KUKA KRL program: FOLGE7.SRC, FOLGE7.DAT

--- FOLGE7.SRC ---
&COMMENT vymena cepicek
&ACCESS RV
&PARAM TPVW_VERSION=3.3.5
DEF FOLGE7 ( )
; FOLD ;%{H} %MKUKATPVW
SPS_N=-1
VW (#VW_AUE_INIT,TRUE)
PENTER:
INTERRUPT DECL 10 WHEN $CYCFLAG[30]==FALSE DO VW(#FB_STOP,TRUE)
INTERRUPT ON 10
INT10=TRUE
; ENDFOLD
;FOLD PTP VB=100% VE=0% ACC=100% Wzg=1 SPSTrig=0[1/100s] FP;%{P}%MKUKATPVW,%CMOVE,%VPTP,%P 1:1, 2: VB=, 3:100, 4:%, 5: VE=, 6:0, 7:%, 8: ACC=, 9:100, 10:%, 11: Wzg=, 12:1, 13: SPSTrig=, 14:0, 15:[1/100s], 16: FP, 17:0, 18:-1, 19:1
; FOLD FB ONL = EIN;%{SE}%MKUKATPVW %CVW_SPS %VFB %P 2:FB ONL = EIN,3:                  FB
;ENDFOLD
;FOLD 1:  SPSMAKRO99 = !F100;%{SE}%MKUKATPVW %CVW_SPS %VMAKRO %P 2:SPSMAKRO99 = !F100,3:             MAKRO
;ENDFOLD
;FOLD 2:  SPSMAKRO96 = EIN;%{SE}%MKUKATPVW %CVW_SPS %VMAKRO %P 2:SPSMAKRO96 = EIN,3:               MAKRO
;ENDFOLD
;FOLD 3:  SPSMAKRO81 = EIN;%{SE}%MKUKATPVW %CVW_SPS %VMAKRO %P 2:SPSMAKRO81 = EIN,3:            MAKRO
;ENDFOLD
;FOLD 4:  SPSMAKRO82 = EIN;%{SE}%MKUKATPVW %CVW_SPS %VMAKRO %P 2:SPSMAKRO82 = EIN,3:           MAKRO
;ENDFOLD
;FOLD 5:  SPSMAKRO95 = EIN;%{SE}%MKUKATPVW %CVW_SPS %VMAKRO %P 2:SPSMAKRO95 = EIN,3:                 MAKRO
;ENDFOLD
;FOLD 6:  bin1 ( EIN ) = 9931;%{SE}%MKUKATPVW %CVW_SPS %VARIASG %P 2:bin1 ( EIN ) = 9931,3:          ARIASG
;ENDFOLD
;FOLD 7:  SPSMAKRO3 = EIN;%{SE}%MKUKATPVW %CVW_SPS %VMAKRO %P 2:SPSMAKRO3 = EIN,3:         MAKRO
;ENDFOLD
;FOLD {H}
SPS_FERTIG = FALSE
INTERRUPT DECL 10 WHEN $CYCFLAG[30]==FALSE DO VW(#FB_STOP,TRUE)
INTERRUPT ON 10
INT10=TRUE
VW(#VW_INIT,TRUE)
VW_USR_R (#USR_INIT)
TRIGGER  WHEN DISTANCE=1 DELAY=-0.1 DO P0_MERKER=TRUE
VW_MPARA_ACT = P0_D
VW(#MPARA,TRUE)
SPS_FERTIG=FALSE
TRIGGER WHEN DISTANCE=1 DELAY=0 DO SPS_TRIG(1) PRIO=-1
TRIGGER WHEN DISTANCE=0 DELAY=0 DO $CYCFLAG[30]=(TRUE) AND $CYCFLAG[31] OR ($TIMER[15]<0)
TRIGGER WHEN DISTANCE=0 DELAY=0 DO $CYC_DEF30[]=" EIN "
PTP P0
WAIT FOR SPS_FERTIG
;ENDFOLD
;ENDFOLD
; FOLD Warte auf Folgenstart ;%{SE}%MKUKATPVW,%C,%V
VW (#VW_AUE_WAIT,TRUE )
IF N_VW==TRUE THEN
GOTO PEXIT
ENDIF
;ENDFOLD
;FOLD PTP VB=100% VE=0% ACC=100% Wzg=1 SPSTrig=0[1/100s] FP;%{P}%MKUKATPVW,%CMOVE,%VPTP,%P 1:1, 2: VB=, 3:100, 4:%, 5: VE=, 6:0, 7:%, 8: ACC=, 9:100, 10:%, 11: Wzg=, 12:1, 13: SPSTrig=, 14:0, 15:[1/100s], 16: FP, 17:1, 18:-1, 19:2
; FOLD FB ONL = EIN;%{SE}%MKUKATPVW %CVW_SPS %VFB %P 2:FB ONL = EIN,3:           FB
;ENDFOLD
;FOLD 1:  F100 = AUS;%{SE}%MKUKATPVW %CVW_SPS %VBOASG %P 2:F100 = AUS,3:          BOASG
;ENDFOLD
;FOLD 2:  F199 = EIN;%{SE}%MKUKATPVW %CVW_SPS %VBOASG %P 2:F199 = EIN,3:         BOASG
;ENDFOLD
;FOLD 3:  SPSMAKRO21 = EIN;%{SE}%MKUKATPVW %CVW_SPS %VMAKRO %P 2:SPSMAKRO21 = EIN,3:        MAKRO
;ENDFOLD
;FOLD 4:  t1 ( EIN ) = 0[1/10Sek];%{SE}%MKUKATPVW %CVW_SPS %VTASG %P 2:t1 ( EIN ) = 0[1/10Sek],3:       TASG
;ENDFOLD
;FOLD {H}
VW_MPARA_ACT = P1_D
VW(#MPARA,TRUE)
SPS_FERTIG=FALSE
TRIGGER WHEN DISTANCE=1 DELAY=0 DO SPS_TRIG(2) PRIO=-1
TRIGGER WHEN DISTANCE=0 DELAY=0 DO $CYCFLAG[30]=(TRUE) AND $CYCFLAG[31] OR ($TIMER[15]<0)
TRIGGER WHEN DISTANCE=0 DELAY=0 DO $CYC_DEF30[]=" EIN "
PTP P1
WAIT FOR SPS_FERTIG
;ENDFOLD
;ENDFOLD
;FOLD PTP VB=100% VE=0% ACC=100% Wzg=1 SPSTrig=0[1/100s] FU;%{P}%MKUKATPVW,%CMOVE,%VPTP,%P 1:1, 2: VB=, 3:100, 4:%, 5: VE=, 6:0, 7:%, 8: ACC=, 9:100, 10:%, 11: Wzg=, 12:1, 13: SPSTrig=, 14:0, 15:[1/100s], 16: FU, 17:3, 18:-1, 19:-1
; FOLD FB ONL = M1;%{SE}%MKUKATPVW %CVW_SPS %VFB %P 2:FB ONL = M1,3:          FB
;ENDFOLD
; FOLD UP8 = F409;%{SE}%MKUKATPVW %CVW_SPS %VUP %P 2:UP8 = F409,3:       UP
;ENDFOLD
; FOLD UP1 = E67 + F401;%{SE}%MKUKATPVW %CVW_SPS %VUP %P 2:UP1 = E67 + F401,3:        UP
;ENDFOLD
;FOLD {H}
VW_MPARA_ACT = P3_D
VW(#MPARA,TRUE)
TRIGGER WHEN DISTANCE=0 DELAY=0 DO $CYCFLAG[30]=($CYCFLAG[1]) AND $CYCFLAG[31] OR ($TIMER[15]<0)
TRIGGER WHEN DISTANCE=0 DELAY=0 DO $CYC_DEF30[]="M1"
PTP P3
WAIT FOR TRUE
SELECT(#UP,8,$FLAG[409])
SELECT(#UP,1,$IN[67] OR $FLAG[401])
;ENDFOLD
;ENDFOLD
;FOLD PTP VB=100% VE=0% ACC=100% Wzg=1 SPSTrig=0[1/100s] FP;%{P}%MKUKATPVW,%CMOVE,%VPTP,%P 1:1, 2: VB=, 3:100, 4:%, 5: VE=, 6:0, 7:%, 8: ACC=, 9:100, 10:%, 11: Wzg=, 12:1, 13: SPSTrig=, 14:0, 15:[1/100s], 16: FP, 17:2, 18:-1, 19:3
; FOLD FB ONL = EIN;%{SE}%MKUKATPVW %CVW_SPS %VFB %P 2:FB ONL = EIN,3:             FB
;ENDFOLD
;FOLD 1:  F100 = EIN;%{SE}%MKUKATPVW %CVW_SPS %VBOASG %P 2:F100 = EIN,3:            BOASG
;ENDFOLD
;FOLD 2:  F199 = AUS;%{SE}%MKUKATPVW %CVW_SPS %VBOASG %P 2:F199 = AUS,3:         BOASG
;ENDFOLD
;FOLD 3:  t1 ( EIN ) = STOP;%{SE}%MKUKATPVW %CVW_SPS %VTSTOP %P 2:t1 ( EIN ) = STOP,3:        TSTOP
;ENDFOLD
;FOLD 4:  t2 ( EIN ) = t1[1/10Sek];%{SE}%MKUKATPVW %CVW_SPS %VTASG %P 2:t2 ( EIN ) = t1[1/10Sek],3:        TASG
;ENDFOLD
;FOLD 5:  t2 ( EIN ) = STOP;%{SE}%MKUKATPVW %CVW_SPS %VTSTOP %P 2:t2 ( EIN ) = STOP,3:       TSTOP
;ENDFOLD
;FOLD 6:  SPSMAKRO81 = EIN;%{SE}%MKUKATPVW %CVW_SPS %VMAKRO %P 2:SPSMAKRO81 = EIN,3:           MAKRO
;ENDFOLD
;FOLD 7:  SPSMAKRO82 = EIN;%{SE}%MKUKATPVW %CVW_SPS %VMAKRO %P 2:SPSMAKRO82 = EIN,3:          MAKRO
;ENDFOLD
;FOLD {H}
VW_MPARA_ACT = P2_D
VW(#MPARA,TRUE)
SPS_FERTIG=FALSE
TRIGGER WHEN DISTANCE=1 DELAY=0 DO SPS_TRIG(3) PRIO=-1
TRIGGER WHEN DISTANCE=0 DELAY=0 DO $CYCFLAG[30]=(TRUE) AND $CYCFLAG[31] OR ($TIMER[15]<0)
TRIGGER WHEN DISTANCE=0 DELAY=0 DO $CYC_DEF30[]=" EIN "
PTP P2
WAIT FOR SPS_FERTIG
;ENDFOLD
;ENDFOLD
; FOLD ;%{H}
VW (#VW_AUE_END,TRUE)
GOTO PENTER
PEXIT:
END
DEF  SPS_TRIG (NO:IN )
INT NO
BOOL UES
IF NO>10000 THEN
NO=NO-10000
UES=TRUE
ELSE
UES=FALSE
ENDIF
IF $PRO_MODE==#MSTEP THEN
IF $PRO_MOVE THEN
WAIT FOR NOT $PRO_MOVE
HALT
ENDIF
ENDIF
SWITCH  NO
CASE 1
;FOLD SPS_TRIG1 {H}
SELECT(#MAKRO,99,NOT $FLAG[100])
SELECT(#MAKRO,96,TRUE)
SELECT(#MAKRO,81,TRUE)
SELECT(#MAKRO,82,TRUE)
SELECT(#MAKRO,95,TRUE)
VW(#BINOUT,TRUE,1,9931)
SELECT(#MAKRO,3,TRUE)
;ENDFOLD
CASE 2
;FOLD SPS_TRIG2 {H}
$FLAG[100]=FALSE
$FLAG[199]=TRUE
SELECT(#MAKRO,21,TRUE)
VW(#SET_TIME,TRUE,1,0,0)
;ENDFOLD
CASE 3
;FOLD SPS_TRIG3 {H}
$FLAG[100]=TRUE
$FLAG[199]=FALSE
VW(#SET_TIME,TRUE,1,1,0)
VW(#SET_TIME,TRUE,2,0,$TIMER[1]*0.01)
VW(#SET_TIME,TRUE,2,1,0)
SELECT(#MAKRO,81,TRUE)
SELECT(#MAKRO,82,TRUE)
;ENDFOLD
CASE 4
;FOLD SPS_TRIG4 {H}
;ENDFOLD
CASE 5
;FOLD SPS_TRIG5 {H}
;ENDFOLD
CASE 6
;FOLD SPS_TRIG6 {H}
;ENDFOLD
CASE 7
;FOLD SPS_TRIG7 {H}
;ENDFOLD
CASE 8
;FOLD SPS_TRIG8 {H}
;ENDFOLD
CASE 9
;FOLD SPS_TRIG9 {H}
;ENDFOLD
CASE 10
;FOLD SPS_TRIG10 {H}
;ENDFOLD
CASE 11
;FOLD SPS_TRIG11 {H}
;ENDFOLD
CASE 12
;FOLD SPS_TRIG12 {H}
;ENDFOLD
CASE 13
;FOLD SPS_TRIG13 {H}
;ENDFOLD
CASE 14
;FOLD SPS_TRIG14 {H}
;ENDFOLD
CASE 15
;FOLD SPS_TRIG15 {H}
;ENDFOLD
CASE 16
;FOLD SPS_TRIG16 {H}
;ENDFOLD
CASE 17
;FOLD SPS_TRIG17 {H}
;ENDFOLD
CASE 18
;FOLD SPS_TRIG18 {H}
;ENDFOLD
CASE 19
;FOLD SPS_TRIG19 {H}
;ENDFOLD
CASE 20
;FOLD SPS_TRIG20 {H}
;ENDFOLD
CASE 21
;FOLD SPS_TRIG21 {H}
;ENDFOLD
CASE 22
;FOLD SPS_TRIG22 {H}
;ENDFOLD
CASE 23
;FOLD SPS_TRIG23 {H}
;ENDFOLD
CASE 24
;FOLD SPS_TRIG24 {H}
;ENDFOLD
CASE 25
;FOLD SPS_TRIG25 {H}
;ENDFOLD
CASE 26
;FOLD SPS_TRIG26 {H}
;ENDFOLD
CASE 27
;FOLD SPS_TRIG27 {H}
;ENDFOLD
CASE 28
;FOLD SPS_TRIG28 {H}
;ENDFOLD
CASE 29
;FOLD SPS_TRIG29 {H}
;ENDFOLD
CASE 30
;FOLD SPS_TRIG30 {H}
;ENDFOLD
CASE 31
;FOLD SPS_TRIG31 {H}
;ENDFOLD
CASE 32
;FOLD SPS_TRIG32 {H}
;ENDFOLD
CASE 33
;FOLD SPS_TRIG33 {H}
;ENDFOLD
CASE 34
;FOLD SPS_TRIG34 {H}
;ENDFOLD
CASE 35
;FOLD SPS_TRIG35 {H}
;ENDFOLD
CASE 36
;FOLD SPS_TRIG36 {H}
;ENDFOLD
CASE 37
;FOLD SPS_TRIG37 {H}
;ENDFOLD
CASE 38
;FOLD SPS_TRIG38 {H}
;ENDFOLD
CASE 39
;FOLD SPS_TRIG39 {H}
;ENDFOLD
CASE 40
;FOLD SPS_TRIG40 {H}
;ENDFOLD
CASE 41
;FOLD SPS_TRIG41 {H}
;ENDFOLD
CASE 42
;FOLD SPS_TRIG42 {H}
;ENDFOLD
CASE 43
;FOLD SPS_TRIG43 {H}
;ENDFOLD
CASE 44
;FOLD SPS_TRIG44 {H}
;ENDFOLD
CASE 45
;FOLD SPS_TRIG45 {H}
;ENDFOLD
CASE 46
;FOLD SPS_TRIG46 {H}
;ENDFOLD
CASE 47
;FOLD SPS_TRIG47 {H}
;ENDFOLD
CASE 48
;FOLD SPS_TRIG48 {H}
;ENDFOLD
CASE 49
;FOLD SPS_TRIG49 {H}
;ENDFOLD
CASE 50
;FOLD SPS_TRIG50 {H}
;ENDFOLD
CASE 51
;FOLD SPS_TRIG51 {H}
;ENDFOLD
CASE 52
;FOLD SPS_TRIG52 {H}
;ENDFOLD
CASE 53
;FOLD SPS_TRIG53 {H}
;ENDFOLD
CASE 54
;FOLD SPS_TRIG54 {H}
;ENDFOLD
CASE 55
;FOLD SPS_TRIG55 {H}
;ENDFOLD
CASE 56
;FOLD SPS_TRIG56 {H}
;ENDFOLD
CASE 57
;FOLD SPS_TRIG57 {H}
;ENDFOLD
CASE 58
;FOLD SPS_TRIG58 {H}
;ENDFOLD
CASE 59
;FOLD SPS_TRIG59 {H}
;ENDFOLD
CASE 60
;FOLD SPS_TRIG60 {H}
;ENDFOLD
CASE 61
;FOLD SPS_TRIG61 {H}
;ENDFOLD
CASE 62
;FOLD SPS_TRIG62 {H}
;ENDFOLD
CASE 63
;FOLD SPS_TRIG63 {H}
;ENDFOLD
CASE 64
;FOLD SPS_TRIG64 {H}
;ENDFOLD
CASE 65
;FOLD SPS_TRIG65 {H}
;ENDFOLD
CASE 66
;FOLD SPS_TRIG66 {H}
;ENDFOLD
CASE 67
;FOLD SPS_TRIG67 {H}
;ENDFOLD
CASE 68
;FOLD SPS_TRIG68 {H}
;ENDFOLD
CASE 69
;FOLD SPS_TRIG69 {H}
;ENDFOLD
CASE 70
;FOLD SPS_TRIG70 {H}
;ENDFOLD
CASE 71
;FOLD SPS_TRIG71 {H}
;ENDFOLD
CASE 72
;FOLD SPS_TRIG72 {H}
;ENDFOLD
CASE 73
;FOLD SPS_TRIG73 {H}
;ENDFOLD
CASE 74
;FOLD SPS_TRIG74 {H}
;ENDFOLD
CASE 75
;FOLD SPS_TRIG75 {H}
;ENDFOLD
CASE 76
;FOLD SPS_TRIG76 {H}
;ENDFOLD
CASE 77
;FOLD SPS_TRIG77 {H}
;ENDFOLD
CASE 78
;FOLD SPS_TRIG78 {H}
;ENDFOLD
CASE 79
;FOLD SPS_TRIG79 {H}
;ENDFOLD
CASE 80
;FOLD SPS_TRIG80 {H}
;ENDFOLD
CASE 81
;FOLD SPS_TRIG81 {H}
;ENDFOLD
CASE 82
;FOLD SPS_TRIG82 {H}
;ENDFOLD
CASE 83
;FOLD SPS_TRIG83 {H}
;ENDFOLD
CASE 84
;FOLD SPS_TRIG84 {H}
;ENDFOLD
CASE 85
;FOLD SPS_TRIG85 {H}
;ENDFOLD
CASE 86
;FOLD SPS_TRIG86 {H}
;ENDFOLD
CASE 87
;FOLD SPS_TRIG87 {H}
;ENDFOLD
CASE 88
;FOLD SPS_TRIG88 {H}
;ENDFOLD
CASE 89
;FOLD SPS_TRIG89 {H}
;ENDFOLD
CASE 90
;FOLD SPS_TRIG90 {H}
;ENDFOLD
CASE 91
;FOLD SPS_TRIG91 {H}
;ENDFOLD
CASE 92
;FOLD SPS_TRIG92 {H}
;ENDFOLD
CASE 93
;FOLD SPS_TRIG93 {H}
;ENDFOLD
CASE 94
;FOLD SPS_TRIG94 {H}
;ENDFOLD
CASE 95
;FOLD SPS_TRIG95 {H}
;ENDFOLD
CASE 96
;FOLD SPS_TRIG96 {H}
;ENDFOLD
CASE 97
;FOLD SPS_TRIG97 {H}
;ENDFOLD
CASE 98
;FOLD SPS_TRIG98 {H}
;ENDFOLD
CASE 99
;FOLD SPS_TRIG99 {H}
;ENDFOLD
CASE 100
;FOLD SPS_TRIG100 {H}
;ENDFOLD
CASE 101
;FOLD SPS_TRIG101 {H}
;ENDFOLD
CASE 102
;FOLD SPS_TRIG102 {H}
;ENDFOLD
CASE 103
;FOLD SPS_TRIG103 {H}
;ENDFOLD
CASE 104
;FOLD SPS_TRIG104 {H}
;ENDFOLD
CASE 105
;FOLD SPS_TRIG105 {H}
;ENDFOLD
CASE 106
;FOLD SPS_TRIG106 {H}
;ENDFOLD
CASE 107
;FOLD SPS_TRIG107 {H}
;ENDFOLD
CASE 108
;FOLD SPS_TRIG108 {H}
;ENDFOLD
CASE 109
;FOLD SPS_TRIG109 {H}
;ENDFOLD
CASE 110
;FOLD SPS_TRIG110 {H}
;ENDFOLD
CASE 111
;FOLD SPS_TRIG111 {H}
;ENDFOLD
CASE 112
;FOLD SPS_TRIG112 {H}
;ENDFOLD
CASE 113
;FOLD SPS_TRIG113 {H}
;ENDFOLD
CASE 114
;FOLD SPS_TRIG114 {H}
;ENDFOLD
CASE 115
;FOLD SPS_TRIG115 {H}
;ENDFOLD
CASE 116
;FOLD SPS_TRIG116 {H}
;ENDFOLD
CASE 117
;FOLD SPS_TRIG117 {H}
;ENDFOLD
CASE 118
;FOLD SPS_TRIG118 {H}
;ENDFOLD
CASE 119
;FOLD SPS_TRIG119 {H}
;ENDFOLD
CASE 120
;FOLD SPS_TRIG120 {H}
;ENDFOLD
CASE 121
;FOLD SPS_TRIG121 {H}
;ENDFOLD
CASE 122
;FOLD SPS_TRIG122 {H}
;ENDFOLD
CASE 123
;FOLD SPS_TRIG123 {H}
;ENDFOLD
CASE 124
;FOLD SPS_TRIG124 {H}
;ENDFOLD
CASE 125
;FOLD SPS_TRIG125 {H}
;ENDFOLD
CASE 126
;FOLD SPS_TRIG126 {H}
;ENDFOLD
CASE 127
;FOLD SPS_TRIG127 {H}
;ENDFOLD
CASE 128
;FOLD SPS_TRIG128 {H}
;ENDFOLD
CASE 129
;FOLD SPS_TRIG129 {H}
;ENDFOLD
CASE 130
;FOLD SPS_TRIG130 {H}
;ENDFOLD
CASE 131
;FOLD SPS_TRIG131 {H}
;ENDFOLD
CASE 132
;FOLD SPS_TRIG132 {H}
;ENDFOLD
CASE 133
;FOLD SPS_TRIG133 {H}
;ENDFOLD
CASE 134
;FOLD SPS_TRIG134 {H}
;ENDFOLD
CASE 135
;FOLD SPS_TRIG135 {H}
;ENDFOLD
CASE 136
;FOLD SPS_TRIG136 {H}
;ENDFOLD
CASE 137
;FOLD SPS_TRIG137 {H}
;ENDFOLD
CASE 138
;FOLD SPS_TRIG138 {H}
;ENDFOLD
CASE 139
;FOLD SPS_TRIG139 {H}
;ENDFOLD
CASE 140
;FOLD SPS_TRIG140 {H}
;ENDFOLD
CASE 141
;FOLD SPS_TRIG141 {H}
;ENDFOLD
CASE 142
;FOLD SPS_TRIG142 {H}
;ENDFOLD
CASE 143
;FOLD SPS_TRIG143 {H}
;ENDFOLD
CASE 144
;FOLD SPS_TRIG144 {H}
;ENDFOLD
CASE 145
;FOLD SPS_TRIG145 {H}
;ENDFOLD
CASE 146
;FOLD SPS_TRIG146 {H}
;ENDFOLD
CASE 147
;FOLD SPS_TRIG147 {H}
;ENDFOLD
CASE 148
;FOLD SPS_TRIG148 {H}
;ENDFOLD
CASE 149
;FOLD SPS_TRIG149 {H}
;ENDFOLD
CASE 150
;FOLD SPS_TRIG150 {H}
;ENDFOLD
CASE 151
;FOLD SPS_TRIG151 {H}
;ENDFOLD
CASE 152
;FOLD SPS_TRIG152 {H}
;ENDFOLD
CASE 153
;FOLD SPS_TRIG153 {H}
;ENDFOLD
CASE 154
;FOLD SPS_TRIG154 {H}
;ENDFOLD
CASE 155
;FOLD SPS_TRIG155 {H}
;ENDFOLD
CASE 156
;FOLD SPS_TRIG156 {H}
;ENDFOLD
CASE 157
;FOLD SPS_TRIG157 {H}
;ENDFOLD
CASE 158
;FOLD SPS_TRIG158 {H}
;ENDFOLD
CASE 159
;FOLD SPS_TRIG159 {H}
;ENDFOLD
CASE 160
;FOLD SPS_TRIG160 {H}
;ENDFOLD
CASE 161
;FOLD SPS_TRIG161 {H}
;ENDFOLD
CASE 162
;FOLD SPS_TRIG162 {H}
;ENDFOLD
CASE 163
;FOLD SPS_TRIG163 {H}
;ENDFOLD
CASE 164
;FOLD SPS_TRIG164 {H}
;ENDFOLD
CASE 165
;FOLD SPS_TRIG165 {H}
;ENDFOLD
CASE 166
;FOLD SPS_TRIG166 {H}
;ENDFOLD
CASE 167
;FOLD SPS_TRIG167 {H}
;ENDFOLD
CASE 168
;FOLD SPS_TRIG168 {H}
;ENDFOLD
CASE 169
;FOLD SPS_TRIG169 {H}
;ENDFOLD
CASE 170
;FOLD SPS_TRIG170 {H}
;ENDFOLD
CASE 171
;FOLD SPS_TRIG171 {H}
;ENDFOLD
CASE 172
;FOLD SPS_TRIG172 {H}
;ENDFOLD
CASE 173
;FOLD SPS_TRIG173 {H}
;ENDFOLD
CASE 174
;FOLD SPS_TRIG174 {H}
;ENDFOLD
CASE 175
;FOLD SPS_TRIG175 {H}
;ENDFOLD
CASE 176
;FOLD SPS_TRIG176 {H}
;ENDFOLD
CASE 177
;FOLD SPS_TRIG177 {H}
;ENDFOLD
CASE 178
;FOLD SPS_TRIG178 {H}
;ENDFOLD
CASE 179
;FOLD SPS_TRIG179 {H}
;ENDFOLD
CASE 180
;FOLD SPS_TRIG180 {H}
;ENDFOLD
CASE 181
;FOLD SPS_TRIG181 {H}
;ENDFOLD
CASE 182
;FOLD SPS_TRIG182 {H}
;ENDFOLD
CASE 183
;FOLD SPS_TRIG183 {H}
;ENDFOLD
CASE 184
;FOLD SPS_TRIG184 {H}
;ENDFOLD
CASE 185
;FOLD SPS_TRIG185 {H}
;ENDFOLD
CASE 186
;FOLD SPS_TRIG186 {H}
;ENDFOLD
CASE 187
;FOLD SPS_TRIG187 {H}
;ENDFOLD
CASE 188
;FOLD SPS_TRIG188 {H}
;ENDFOLD
CASE 189
;FOLD SPS_TRIG189 {H}
;ENDFOLD
CASE 190
;FOLD SPS_TRIG190 {H}
;ENDFOLD
CASE 191
;FOLD SPS_TRIG191 {H}
;ENDFOLD
CASE 192
;FOLD SPS_TRIG192 {H}
;ENDFOLD
CASE 193
;FOLD SPS_TRIG193 {H}
;ENDFOLD
CASE 194
;FOLD SPS_TRIG194 {H}
;ENDFOLD
CASE 195
;FOLD SPS_TRIG195 {H}
;ENDFOLD
CASE 196
;FOLD SPS_TRIG196 {H}
;ENDFOLD
CASE 197
;FOLD SPS_TRIG197 {H}
;ENDFOLD
CASE 198
;FOLD SPS_TRIG198 {H}
;ENDFOLD
CASE 199
;FOLD SPS_TRIG199 {H}
;ENDFOLD
CASE 200
;FOLD SPS_TRIG200 {H}
;ENDFOLD
CASE 201
;FOLD SPS_TRIG201 {H}
;ENDFOLD
CASE 202
;FOLD SPS_TRIG202 {H}
;ENDFOLD
CASE 203
;FOLD SPS_TRIG203 {H}
;ENDFOLD
CASE 204
;FOLD SPS_TRIG204 {H}
;ENDFOLD
CASE 205
;FOLD SPS_TRIG205 {H}
;ENDFOLD
CASE 206
;FOLD SPS_TRIG206 {H}
;ENDFOLD
CASE 207
;FOLD SPS_TRIG207 {H}
;ENDFOLD
CASE 208
;FOLD SPS_TRIG208 {H}
;ENDFOLD
CASE 209
;FOLD SPS_TRIG209 {H}
;ENDFOLD
CASE 210
;FOLD SPS_TRIG210 {H}
;ENDFOLD
CASE 211
;FOLD SPS_TRIG211 {H}
;ENDFOLD
CASE 212
;FOLD SPS_TRIG212 {H}
;ENDFOLD
CASE 213
;FOLD SPS_TRIG213 {H}
;ENDFOLD
CASE 214
;FOLD SPS_TRIG214 {H}
;ENDFOLD
CASE 215
;FOLD SPS_TRIG215 {H}
;ENDFOLD
CASE 216
;FOLD SPS_TRIG216 {H}
;ENDFOLD
CASE 217
;FOLD SPS_TRIG217 {H}
;ENDFOLD
CASE 218
;FOLD SPS_TRIG218 {H}
;ENDFOLD
CASE 219
;FOLD SPS_TRIG219 {H}
;ENDFOLD
CASE 220
;FOLD SPS_TRIG220 {H}
;ENDFOLD
CASE 221
;FOLD SPS_TRIG221 {H}
;ENDFOLD
CASE 222
;FOLD SPS_TRIG222 {H}
;ENDFOLD
CASE 223
;FOLD SPS_TRIG223 {H}
;ENDFOLD
CASE 224
;FOLD SPS_TRIG224 {H}
;ENDFOLD
CASE 225
;FOLD SPS_TRIG225 {H}
;ENDFOLD
CASE 226
;FOLD SPS_TRIG226 {H}
;ENDFOLD
CASE 227
;FOLD SPS_TRIG227 {H}
;ENDFOLD
CASE 228
;FOLD SPS_TRIG228 {H}
;ENDFOLD
CASE 229
;FOLD SPS_TRIG229 {H}
;ENDFOLD
CASE 230
;FOLD SPS_TRIG230 {H}
;ENDFOLD
CASE 231
;FOLD SPS_TRIG231 {H}
;ENDFOLD
CASE 232
;FOLD SPS_TRIG232 {H}
;ENDFOLD
CASE 233
;FOLD SPS_TRIG233 {H}
;ENDFOLD
CASE 234
;FOLD SPS_TRIG234 {H}
;ENDFOLD
CASE 235
;FOLD SPS_TRIG235 {H}
;ENDFOLD
CASE 236
;FOLD SPS_TRIG236 {H}
;ENDFOLD
CASE 237
;FOLD SPS_TRIG237 {H}
;ENDFOLD
CASE 238
;FOLD SPS_TRIG238 {H}
;ENDFOLD
CASE 239
;FOLD SPS_TRIG239 {H}
;ENDFOLD
CASE 240
;FOLD SPS_TRIG240 {H}
;ENDFOLD
CASE 241
;FOLD SPS_TRIG241 {H}
;ENDFOLD
CASE 242
;FOLD SPS_TRIG242 {H}
;ENDFOLD
CASE 243
;FOLD SPS_TRIG243 {H}
;ENDFOLD
CASE 244
;FOLD SPS_TRIG244 {H}
;ENDFOLD
CASE 245
;FOLD SPS_TRIG245 {H}
;ENDFOLD
CASE 246
;FOLD SPS_TRIG246 {H}
;ENDFOLD
CASE 247
;FOLD SPS_TRIG247 {H}
;ENDFOLD
CASE 248
;FOLD SPS_TRIG248 {H}
;ENDFOLD
CASE 249
;FOLD SPS_TRIG249 {H}
;ENDFOLD
CASE 250
;FOLD SPS_TRIG250 {H}
;ENDFOLD
CASE 251
;FOLD SPS_TRIG251 {H}
;ENDFOLD
CASE 252
;FOLD SPS_TRIG252 {H}
;ENDFOLD
CASE 253
;FOLD SPS_TRIG253 {H}
;ENDFOLD
CASE 254
;FOLD SPS_TRIG254 {H}
;ENDFOLD
CASE 255
;FOLD SPS_TRIG255 {H}
;ENDFOLD
CASE 256
;FOLD SPS_TRIG256 {H}
;ENDFOLD
CASE 257
;FOLD SPS_TRIG257 {H}
;ENDFOLD
CASE 258
;FOLD SPS_TRIG258 {H}
;ENDFOLD
CASE 259
;FOLD SPS_TRIG259 {H}
;ENDFOLD
CASE 260
;FOLD SPS_TRIG260 {H}
;ENDFOLD
CASE 261
;FOLD SPS_TRIG261 {H}
;ENDFOLD
CASE 262
;FOLD SPS_TRIG262 {H}
;ENDFOLD
CASE 263
;FOLD SPS_TRIG263 {H}
;ENDFOLD
CASE 264
;FOLD SPS_TRIG264 {H}
;ENDFOLD
CASE 265
;FOLD SPS_TRIG265 {H}
;ENDFOLD
CASE 266
;FOLD SPS_TRIG266 {H}
;ENDFOLD
CASE 267
;FOLD SPS_TRIG267 {H}
;ENDFOLD
CASE 268
;FOLD SPS_TRIG268 {H}
;ENDFOLD
CASE 269
;FOLD SPS_TRIG269 {H}
;ENDFOLD
CASE 270
;FOLD SPS_TRIG270 {H}
;ENDFOLD
CASE 271
;FOLD SPS_TRIG271 {H}
;ENDFOLD
CASE 272
;FOLD SPS_TRIG272 {H}
;ENDFOLD
CASE 273
;FOLD SPS_TRIG273 {H}
;ENDFOLD
CASE 274
;FOLD SPS_TRIG274 {H}
;ENDFOLD
CASE 275
;FOLD SPS_TRIG275 {H}
;ENDFOLD
CASE 276
;FOLD SPS_TRIG276 {H}
;ENDFOLD
CASE 277
;FOLD SPS_TRIG277 {H}
;ENDFOLD
CASE 278
;FOLD SPS_TRIG278 {H}
;ENDFOLD
CASE 279
;FOLD SPS_TRIG279 {H}
;ENDFOLD
CASE 280
;FOLD SPS_TRIG280 {H}
;ENDFOLD
CASE 281
;FOLD SPS_TRIG281 {H}
;ENDFOLD
CASE 282
;FOLD SPS_TRIG282 {H}
;ENDFOLD
CASE 283
;FOLD SPS_TRIG283 {H}
;ENDFOLD
CASE 284
;FOLD SPS_TRIG284 {H}
;ENDFOLD
CASE 285
;FOLD SPS_TRIG285 {H}
;ENDFOLD
CASE 286
;FOLD SPS_TRIG286 {H}
;ENDFOLD
CASE 287
;FOLD SPS_TRIG287 {H}
;ENDFOLD
CASE 288
;FOLD SPS_TRIG288 {H}
;ENDFOLD
CASE 289
;FOLD SPS_TRIG289 {H}
;ENDFOLD
CASE 290
;FOLD SPS_TRIG290 {H}
;ENDFOLD
CASE 291
;FOLD SPS_TRIG291 {H}
;ENDFOLD
CASE 292
;FOLD SPS_TRIG292 {H}
;ENDFOLD
CASE 293
;FOLD SPS_TRIG293 {H}
;ENDFOLD
CASE 294
;FOLD SPS_TRIG294 {H}
;ENDFOLD
CASE 295
;FOLD SPS_TRIG295 {H}
;ENDFOLD
CASE 296
;FOLD SPS_TRIG296 {H}
;ENDFOLD
CASE 297
;FOLD SPS_TRIG297 {H}
;ENDFOLD
CASE 298
;FOLD SPS_TRIG298 {H}
;ENDFOLD
CASE 299
;FOLD SPS_TRIG299 {H}
;ENDFOLD
CASE 300
;FOLD SPS_TRIG300 {H}
;ENDFOLD
DEFAULT
ENDSWITCH
IF NOT UES THEN
IF ($PRO_MODE==#MSTEP) THEN
HALT
ENDIF
SPS_FERTIG=TRUE
ENDIF
END
; ENDFOLD

--- FOLGE7.DAT ---
&COMMENT vymena cepicek
&ACCESS RV
&PARAM TPVW_VERSION=3.3.5
DEFDAT FOLGE7
; interface to basic routines
EXT BAS (BAS_COMMAND :IN,REAL :IN )
; interface to VW-standard routines
EXT VW (VW_COMMAND:IN, BOOL: IN, REAL:IN, REAL:IN, REAL:IN, REAL:IN, BOOL :IN, E6POS :IN )
; interface to VW_USER - Call
EXT  VW_USER (VW_USER_CMD :IN,REAL  :IN,REAL  :IN,REAL  :IN,REAL  :IN,REAL  :IN,REAL  :IN,BOOL  :IN )
EXT  VW_USR_R (VW_USER_CMD :IN,REAL  :IN,REAL  :IN,REAL  :IN,REAL  :IN,REAL  :IN,REAL  :IN,BOOL  :IN )
; interface select routine
EXT  SELECT (SUBTYPE  :IN,INT  :IN,BOOL  :IN,ARI_TYP  :IN,INT  :IN,BOOL_TYP  :IN,INT  :IN )
INT VW_NEXT_FREE=4
INT VW_NFREE_SPS=4
INT VW_MAX_SPS=300
DECL VW_MPARA_TYP P0_D={TOOL_NO 1,BASE_NO 0 ,VB 100,VE 0,ACC 100,TRG_TIME 0,MOVE_TYPE #PTP_MOTION}
E6POS P0={x 309.224701,y -149.652298,z 1745.69897,a -77.6275101,b -57.8838997,c -160.022995,s 2,t 34,e1 0.0,e2 0.0,e3 0.0,e4 0.0,e5 0.0,e6 0.0}
DECL VW_MPARA_TYP P1_D={TOOL_NO 1,BASE_NO 0 ,VB 100,VE 0,ACC 100,TRG_TIME 0,MOVE_TYPE #PTP_MOTION}
DECL E6POS P1={x 309.224701,y -149.652298,z 1745.69897,a -77.6275101,b -57.8838997,c -160.022995,s 2,t 34,e1 0.0,e2 0.0,e3 0.0,e4 0.0,e5 0.0,e6 0.0}
DECL VW_MPARA_TYP P2_D={TOOL_NO 1,BASE_NO 0 ,VB 100,VE 0,ACC 100,TRG_TIME 0,MOVE_TYPE #PTP_MOTION}
DECL E6POS P2={x 309.224701,y -149.652298,z 1745.69897,a -77.6275101,b -57.8838997,c -160.022995,s 2,t 34,e1 0.0,e2 0.0,e3 0.0,e4 0.0,e5 0.0,e6 0.0}
DECL VW_MPARA_TYP P3_D={TOOL_NO 1,BASE_NO 0 ,VB 100,VE 0,ACC 100,TRG_TIME 0,MOVE_TYPE #PTP_MOTION}
DECL E6POS P3={x 309.224701,y -149.652298,z 1745.69897,a -77.6275101,b -57.8838997,c -160.022995,s 2,t 34,e1 0.0,e2 0.0,e3 0.0,e4 0.0,e5 0.0,e6 0.0}
ENDDAT
